// TIA Portal V18 export
DATA_BLOCK "Pop-up Db"   // DB341
{ S7_Optimized_Access := 'TRUE' }
VERSION : 0.1
// stored: AutoNumber true, DBAccessibleFromOPCUA true, IsOnlyStoredInLoadMemory false, IsRetainMemResEnabled false, IsWriteProtectedInAS false, MemoryReserve 100
   VAR
      "Additional metering Popup-enable" : Bool;
      "Close Button" : Bool;
      "General Visibility" : Bool;
      "Dearing A Visibility" : Bool;
      "Dearing B Visibility" : Bool;
      "Dearing C Visibility" : Bool;
      "Condition check visibility" : Bool;
   END_VAR
   VAR RETAIN
      parameter_scrno_condchecken : String[2];
   END_VAR
BEGIN
END_DATA_BLOCK
